// TIA Portal V19 export
TYPE "LEXCHANGETRAY_typeXXXIoSignalInterface"
// stored: Access Published
   STRUCT
      configuration : "LEXCHANGETRAY_typeXXXSignalConfigeration";
      commands { S7_SetPoint := 'True'} : "LEXCHANGETRAY_typeXXXIoSignalManualCommands";
      monitoring { S7_SetPoint := 'True'} : "LEXCHANGETRAY_typeXXXIoSignalProcessValues";
   END_STRUCT;
END_TYPE
